// TIA Portal V18 export
DATA_BLOCK "ST10_SafetyGate2_DB"   // DB1142
VERSION : 0.1
// stored: AutoNumber false, DBAccessibleFromOPCUA true, DBAccessibleFromWebserver true, InstanceOfName SafetyGate, InstanceOfType FB
"SafetyGate"
   // VAR_INPUT
   //    iSysInface : "RCS_SysComInterface_V1";
   //    "iSafetyGate Opened Monitor" : Bool;
   //    "iSafetyGate Locked Monitor" : Bool;
   //    i1s_Pulse : Bool;
   //    "iSafetyGate AutoLock Timer" : Time;
   //    "iSafetyGate ManualLock Timer" : Time;
   //    iMode : Int;
   // END_VAR
   // VAR_OUTPUT
   //    "oSafetyGate LockedLamp" { ExternalAccessible := 'False'; ExternalVisible := 'False'; ExternalWritable := 'False'} : Bool;
   // END_VAR
   // VAR_IN_OUT
   //    ioSafetyGateLock : Bool;
   //    ioHMI_Interface : "SafetyGateUDT";
   // END_VAR
   // VAR
   //    "sSafetyGate Timer" { S7_SetPoint := 'True'} : Array[1..5] of TON_TIME;
   //    sP_Trig : Array[1..10] of Bool;
   //    sN_Trig : Array[1..10] of Bool;
   //    "sSafetyGate UnlockRequest" { ExternalAccessible := 'False'; ExternalVisible := 'False'; ExternalWritable := 'False'} : Bool;
   //    "sSafetyGate LockRequest" : Bool;
   // END_VAR
BEGIN
END_DATA_BLOCK
